{attribute addProperty BoxType "EL2819-0000-0016"}
{attribute addProperty Id "DIG_Diag_InputsAT %I*DIG_Diag_Inputs_2815A2556480DIG_Inputs_DeviceAT %I*DIG_Inputs_Device_07359F0E3240DIG_OutputsAT %Q*DIG_Outputs_FCF3AB2C1620WcStateAT %I*WcState_F855686C1620InfoDataAT %I*InfoData_BC63D37F80100"}
{attribute addProperty CRC "1054946678"}
{attribute addProperty SizeInBites "208"}
{attribute addProperty SizeInBytes "26"}
TYPE EL2819_CAFBAEBC :
STRUCT
	{attribute addProperty Name "DIG_Diag_Inputs"}
	DIG_Diag_Inputs : DIG_Diag_Inputs_2815A255;
	{attribute addProperty Name "DIG_Inputs_Device"}
	DIG_Inputs_Device : DIG_Inputs_Device_07359F0E;
	{attribute addProperty Name "DIG_Outputs"}
	DIG_Outputs : DIG_Outputs_FCF3AB2C;
	{attribute addProperty Name "WcState"}
	WcState : WcState_F855686C;
	{attribute addProperty Name "InfoData"}
	InfoData : InfoData_BC63D37F;
END_STRUCT
END_TYPE

(* stored: Version 1.2.0.0, ProductVersion 3.1.4024.9
   DUT EL2819_CAFBAEBC: Id {c3f2df31-bfce-47d7-9db9-db88d61dd14b} *)
